KUKA KRL data list: Work_Data.dat

&ACCESS RV
DEFDAT  WORK_DATA PUBLIC
GLOBAL BOOL Work_1=FALSE
GLOBAL BOOL Work_2=FALSE
GLOBAL BOOL Work_3=FALSE
GLOBAL BOOL Work_4=FALSE
ENDDAT
